// TIA Portal V21 export
// export: Created 2026-07-07T07:59:19.9794854Z, ExportSetting WithReadOnly, DisplayName Totally Integrated Automation Portal, DisplayVersion V21, DisplayName SINAMICS Startdrive Advanced, DisplayVersion V21, DisplayName SINAMICS Startdrive G110M, G120, G120C, G120D, G120P, G115D, DisplayVersion V21, DisplayName SINAMICS Startdrive G130, G150, S120, S150, G200, G220, S200, S210, S220, Innomotics MVD, DisplayVersion V21, DisplayName STEP 7 Professional, DisplayVersion V21, DisplayName STEP 7 Safety, DisplayVersion V21, DisplayName Tech WebApplication, DisplayVersion V21, DisplayName WinCC Basic/Comfort/Advanced, DisplayVersion V21, DisplayName WinCC Professional, DisplayVersion V21, DisplayName WinCC Unified, DisplayVersion V21
FUNCTION "FC_CallFertigationControl" : Void   // FC1, SCL
{ S7_Optimized_Access := 'TRUE' }
// stored: CodeModifiedDate 2026-07-07T07:50:57.6980246Z, CompileDate 2026-07-07T07:50:57.6980246Z, CreationDate 2026-07-07T07:50:54.7797252Z, DownloadDate 2026-07-07T07:57:30.9172103Z, InterfaceModifiedDate 2026-07-07T07:50:54.7797252Z, IsConsistent true, LibraryConformanceStatus 错误： 该块中包含单实例调用。 警告： 该对象包含对全局数据块的访问。, LoadMemoryLength 34740, ModifiedDate 2026-07-07T07:50:57.6980246Z, PLCSimAdvancedSupport true, ParameterModified 2026-07-07T07:50:54.7797252Z, SetENOAutomatically false, StructureModified 2026-07-07T07:50:54.7797252Z, WorkMemoryLength 1915
   VAR_TEMP
      Manual_q_f_target : Real;
      Manual_q_a_target : Real;
      Manual_q_n_target : Real;
      Manual_q_p_target : Real;
      Manual_q_k_target : Real;
   END_VAR
BEGIN

      // 在 OB1 中调用本 FC，即可完成：
      // DB1 输入区 -> FB_FertigationControl -> DB1 输出区。
      // 优先级：急停 > 手动模式 > 自动闭环。

      IF "DB1".Emergency_Stop THEN
         "DB1".Manual_Active := FALSE;
         "DB1".Auto_Active := FALSE;
         "DB1".q_f_cmd := 0.0;
         "DB1".q_a_cmd := 0.0;
         "DB1".q_n_cmd := 0.0;
         "DB1".q_p_cmd := 0.0;
         "DB1".q_k_cmd := 0.0;
         "DB1".Valve_F_Actual := 0.0;
         "DB1".Valve_A_Actual := 0.0;
         "DB1".AQ_Valve_F_Raw := 0;
         "DB1".AQ_Valve_A_Raw := 0;
         "DB1".AQ_Valve_N_Raw := 0;
         "DB1".AQ_Valve_P_Raw := 0;
         "DB1".AQ_Valve_K_Raw := 0;
         "DB1".System_Alarm_Light := TRUE;
         "DB1".Actual_Valve_F := 0.0;
         "DB1".Actual_Valve_A := 0.0;
         "DB1".Valve_F_Opt_SP := 0.0;
         "DB1".Valve_A_Opt_SP := 0.0;
         "DB1".Ramp_Target_F := 0.0;
         "DB1".Ramp_Target_A := 0.0;
         RETURN;
      END_IF;

      IF "DB1".Manual_Mode THEN
         "DB1".Manual_Active := TRUE;
         "DB1".Auto_Active := FALSE;

         #Manual_q_f_target := "DB1".Manual_q_f_Set;
         IF #Manual_q_f_target < 0.0 THEN
            #Manual_q_f_target := 0.0;
         ELSIF #Manual_q_f_target > 10.0 THEN
            #Manual_q_f_target := 10.0;
         END_IF;

         #Manual_q_a_target := "DB1".Manual_q_a_Set;
         IF #Manual_q_a_target < 0.0 THEN
            #Manual_q_a_target := 0.0;
         ELSIF #Manual_q_a_target > 4.0 THEN
            #Manual_q_a_target := 4.0;
         END_IF;

         #Manual_q_n_target := "DB1".Manual_q_n_Set;
         IF #Manual_q_n_target < 0.0 THEN
            #Manual_q_n_target := 0.0;
         ELSIF #Manual_q_n_target > "DB1".N_Max THEN
            #Manual_q_n_target := "DB1".N_Max;
         END_IF;

         #Manual_q_p_target := "DB1".Manual_q_p_Set;
         IF #Manual_q_p_target < 0.0 THEN
            #Manual_q_p_target := 0.0;
         ELSIF #Manual_q_p_target > "DB1".P_Max THEN
            #Manual_q_p_target := "DB1".P_Max;
         END_IF;

         #Manual_q_k_target := "DB1".Manual_q_k_Set;
         IF #Manual_q_k_target < 0.0 THEN
            #Manual_q_k_target := 0.0;
         ELSIF #Manual_q_k_target > "DB1".K_Max THEN
            #Manual_q_k_target := "DB1".K_Max;
         END_IF;

         "inst_RL_F"(
            target := #Manual_q_f_target,
            maxRateUp := 1.5,
            maxRateDown := 2.0,
            cycleTime := 0.1,
            enable := TRUE,
            reset := FALSE,
            output => "DB1".q_f_cmd,
            isLimited => "DB1".q_f_limited
         );

         "inst_RL_A"(
            target := #Manual_q_a_target,
            maxRateUp := 0.40,
            maxRateDown := 0.45,
            cycleTime := 0.1,
            enable := TRUE,
            reset := FALSE,
            output => "DB1".q_a_cmd,
            isLimited => "DB1".q_a_limited
         );

         "DB1".q_n_cmd := #Manual_q_n_target;
         "DB1".q_p_cmd := #Manual_q_p_target;
         "DB1".q_k_cmd := #Manual_q_k_target;
         "DB1".q_f_raw := "DB1".q_f_cmd;
         "DB1".q_a_raw := "DB1".q_a_cmd;
         "DB1".Valve_F_Actual := "DB1".q_f_cmd;
         "DB1".Valve_A_Actual := "DB1".q_a_cmd;
         "DB1".AQ_Valve_F_Raw := REAL_TO_INT("DB1".q_f_cmd / 10.0 * 27648.0);
         "DB1".AQ_Valve_A_Raw := REAL_TO_INT("DB1".q_a_cmd / 4.0 * 27648.0);
         IF "DB1".N_Max > 0.0 THEN
            "DB1".AQ_Valve_N_Raw := REAL_TO_INT("DB1".q_n_cmd / "DB1".N_Max * 27648.0);
         ELSE
            "DB1".AQ_Valve_N_Raw := 0;
         END_IF;
         IF "DB1".P_Max > 0.0 THEN
            "DB1".AQ_Valve_P_Raw := REAL_TO_INT("DB1".q_p_cmd / "DB1".P_Max * 27648.0);
         ELSE
            "DB1".AQ_Valve_P_Raw := 0;
         END_IF;
         IF "DB1".K_Max > 0.0 THEN
            "DB1".AQ_Valve_K_Raw := REAL_TO_INT("DB1".q_k_cmd / "DB1".K_Max * 27648.0);
         ELSE
            "DB1".AQ_Valve_K_Raw := 0;
         END_IF;
         "DB1".System_Alarm_Light := FALSE;
         "DB1".Actual_Valve_F := "DB1".Valve_F_Actual;
         "DB1".Actual_Valve_A := "DB1".Valve_A_Actual;
         "DB1".Valve_F_Opt_SP := "DB1".q_f_cmd;
         "DB1".Valve_A_Opt_SP := "DB1".q_a_cmd;
         "DB1".Ramp_Target_F := "DB1".q_f_cmd;
         "DB1".Ramp_Target_A := "DB1".q_a_cmd;
         RETURN;
      END_IF;

      "DB1".Manual_Active := FALSE;
      "DB1".Auto_Active := TRUE;

      IF "DB1".Stage_Auto_SP_Enable AND NOT "DB1".SAC_Enable THEN
         IF "DB1".Growth_Stage = 0 THEN
            "DB1".EC_Set_SP := 0.8;
            "DB1".pH_Set_SP := 6.2;
         ELSIF "DB1".Growth_Stage = 1 THEN
            "DB1".EC_Set_SP := 1.1;
            "DB1".pH_Set_SP := 6.1;
         ELSIF "DB1".Growth_Stage = 2 THEN
            "DB1".EC_Set_SP := 1.5;
            "DB1".pH_Set_SP := 5.9;
         ELSE
            "DB1".EC_Set_SP := 1.0;
            "DB1".pH_Set_SP := 6.1;
         END_IF;
      END_IF;

      "inst_FertigationControl"(
         EC_Set_SP := "DB1".EC_Set_SP,
         pH_Set_SP := "DB1".pH_Set_SP,
         EC_Actual := "DB1".EC_Actual,
         pH_Actual := "DB1".pH_Actual,
         SAC_Enable := "DB1".SAC_Enable,
         Remote_Heartbeat := "DB1".Remote_Heartbeat,
         CycleTime := 0.1,
         Kp_EC := "DB1".Kp_EC_Set,
         Ki_EC := "DB1".Ki_EC_Set,
         Kd_EC := "DB1".Kd_EC_Set,
         Kp_pH := "DB1".Kp_pH_Set,
         Ki_pH := "DB1".Ki_pH_Set,
         Kd_pH := "DB1".Kd_pH_Set,
         EC_Filter_Tau := 2.0,
         pH_Filter_Tau := 4.0,
         EC_Deadband := 0.03,
         pH_Deadband := 0.06,
         EC_Trim_Band := "DB1".EC_Trim_Band,
         pH_Trim_Band := "DB1".pH_Trim_Band,
         EC_MaxInputStep := 0.15,
         pH_MaxInputStep := 0.10,
         q_f_min := 0.0,
         q_f_max := 10.0,
         q_a_min := 0.0,
         q_a_max := 4.0,
         N_Enable := "DB1".N_Enable,
         N_Ratio := "DB1".N_Ratio,
         N_Target := "DB1".N_Target,
         N_Actual := "DB1".N_Actual,
         Kp_N := "DB1".Kp_N_Set,
         Ki_N := "DB1".Ki_N_Set,
         Kd_N := "DB1".Kd_N_Set,
         N_Max := "DB1".N_Max,
         P_Enable := "DB1".P_Enable,
         P_Ratio := "DB1".P_Ratio,
         P_Target := "DB1".P_Target,
         P_Actual := "DB1".P_Actual,
         Kp_P := "DB1".Kp_P_Set,
         Ki_P := "DB1".Ki_P_Set,
         Kd_P := "DB1".Kd_P_Set,
         P_Max := "DB1".P_Max,
         K_Enable := "DB1".K_Enable,
         K_Ratio := "DB1".K_Ratio,
         K_Target := "DB1".K_Target,
         K_Actual := "DB1".K_Actual,
         Kp_K := "DB1".Kp_K_Set,
         Ki_K := "DB1".Ki_K_Set,
         Kd_K := "DB1".Kd_K_Set,
         K_Max := "DB1".K_Max,
         Watchdog_Limit := 10000,
         Growth_Stage := "DB1".Growth_Stage,
         Remote_Comms_OK => "DB1".Remote_Comms_OK,
         Watchdog_Timer => "DB1".Watchdog_Timer,
         Stage_EC_SP => "DB1".Stage_EC_SP,
         Stage_pH_SP => "DB1".Stage_pH_SP,
         Active_EC_SP => "DB1".Active_EC_SP,
         Active_pH_SP => "DB1".Active_pH_SP,
         Setpoint_Protection_Active => "DB1".Setpoint_Protection_Active,
         q_f_cmd => "DB1".q_f_cmd,
         q_a_cmd => "DB1".q_a_cmd,
         Valve_F_Actual => "DB1".Valve_F_Actual,
         Valve_A_Actual => "DB1".Valve_A_Actual,
         AQ_Valve_F_Raw => "DB1".AQ_Valve_F_Raw,
         AQ_Valve_A_Raw => "DB1".AQ_Valve_A_Raw,
         q_n_cmd => "DB1".q_n_cmd,
         q_p_cmd => "DB1".q_p_cmd,
         q_k_cmd => "DB1".q_k_cmd,
         AQ_Valve_N_Raw => "DB1".AQ_Valve_N_Raw,
         AQ_Valve_P_Raw => "DB1".AQ_Valve_P_Raw,
         AQ_Valve_K_Raw => "DB1".AQ_Valve_K_Raw,
         System_Alarm_Light => "DB1".System_Alarm_Light
      );

      // 同步部分内部状态到 DB1，方便在线监控。
      "DB1".Last_Heartbeat := "inst_FertigationControl".Last_Heartbeat;
      "DB1".Watchdog_Count := "inst_FertigationControl".Watchdog_Count;
      "DB1".q_f_raw := "inst_FertigationControl".q_f_raw;
      "DB1".q_a_raw := "inst_FertigationControl".q_a_raw;

      // 兼容旧变量名，若旧监控画面或旧网络还在看 Actual_Valve_F/A，
      // 这里同步为当前 B 方案执行层输出。
      "DB1".Actual_Valve_F := "DB1".Valve_F_Actual;
      "DB1".Actual_Valve_A := "DB1".Valve_A_Actual;
      "DB1".Valve_F_Opt_SP := "DB1".q_f_cmd;
      "DB1".Valve_A_Opt_SP := "DB1".q_a_cmd;
      "DB1".Ramp_Target_F := "DB1".q_f_cmd;
      "DB1".Ramp_Target_A := "DB1".q_a_cmd;
      "DB1".Remote_Comms_Was_OK := "DB1".Remote_Comms_OK;
END_FUNCTION
